INTERFACE OpenDichtSchuif

METHOD Dicht
VAR_INPUT
END_VAR
END_METHOD

METHOD Open
VAR_INPUT
END_VAR
END_METHOD

PROPERTY OpenDichtSchuifStatus : EOpenDichtSchuifStatus
GET
END_GET
SET
END_SET
END_PROPERTY

END_INTERFACE

(* stored: Version 1.1.0.1
   Itf OpenDichtSchuif: Id {0e02246c-75de-4a4d-9082-21ffa56f144a}
   Method Dicht: Id {2967d8ea-a688-47a5-9d7b-f47d16a1b381}
   Method Open: Id {5ebdbeb3-8def-43b4-9074-589eceb818f8}
   Property OpenDichtSchuifStatus: Id {a434d457-9ef9-4311-be43-68dd2d55a58a}
   Get Get: Id {79ff863a-dd76-472a-912f-5e294bc5da9b}
   Set Set: Id {2568d9c7-aa37-41ad-8152-af3ce461868c} *)
